FUNCTION_BLOCK FB_OpenLoopControl
VAR_INPUT
	bEnable: BOOL;
	fInput_ms: LREAL;
	stParam : ST_Parameters;
END_VAR
VAR_OUTPUT
	fNormalizedOutput: LREAL;
END_VAR
VAR
	fFlowReference_m3s : LREAL;
	fM3sToLmin : LREAL := 60000;
END_VAR

IF fInput_ms >= 0.0 THEN 
    fFlowReference_m3s := stparam.stOpenLoopControl.fBoreArea * fInput_ms;
ELSE 
    fFlowReference_m3s := fInput_ms * stparam.stOpenLoopControl.fAnnulusArea;
END_IF;

IF bEnable THEN 
    fNormalizedOutput := (fM3sToLmin * fFlowReference_m3s) / stParam.stOpenLoopControl.fMaxFlowCapacity;
ELSE 
    fNormalizedOutput := 0.0;
END_IF;

IF fNormalizedOutput > 1.0 THEN 
    fNormalizedOutput := 1.0;
ELSIF fNormalizedOutput < -1.0 THEN 
    fNormalizedOutput := -1.0;
END_IF;

END_FUNCTION_BLOCK

(* stored: Version 1.1.0.1, ProductVersion 3.1.4024.10
   POU FB_OpenLoopControl: Id {f423ba7b-c166-485b-8b1a-777fcd38eb4f}, SpecialFunc None *)
